PROGRAM MAIN
VAR
END_VAR

(* 
	GOF 		Define a one-to-many dependency between objects so that when one object changes state, 
				all its dependents are notified and updated automatically   
*)
P_ObserverPattern();

END_PROGRAM

(* stored: Version 1.1.0.1, ProductVersion 3.1.4024.12
   POU MAIN: Id {89ccf36b-f341-4421-bd55-3f0b5179fcd6}, SpecialFunc None *)
